PROGRAM FlyingSaw
VAR
	fbAxisSync : AxisSync; //we initialize the function block that does all the logic
	
	bReset : BOOL; //bool variable connected to a button in the HMI
	bMove : BOOL; //bool variable connected to a button in the HMI
	
	bSensor : BOOL; //bool variable connected to a light in the HMI (turns on when the sync process starts)
	
	rMasterPosition : LREAL; //LREAL variables that display the position of the motors
	rSlavePosition : LREAL;
END_VAR

fbAxisSync.bButton := bMove; //we connect all the variables to the variables of the function block accordingly
fbAxisSync.bResetButton := bReset;

bSensor := fbAxisSync.bSyncSensor;

rMasterPosition := fbAxisSync.rMasterPos;
rSlavePosition := fbAxisSync.rSlavePos;

fbAxisSync(); //we call the funciton block

END_PROGRAM

(* stored: Version 1.1.0.1, ProductVersion 3.1.4024.12
   POU FlyingSaw: Id {066969ca-edf5-450c-bcfd-d777d82ac11b}, SpecialFunc None *)
